(* CODESYS project testPrj.project
   Title: testPrj
   Version: 0.0.0.0

Project tree, tasks and I/O mapping:
  MyController : TM241CE40R, Schneider Electric, order no. TM241CE40R, version 4.0.2.20
    application Application
      libraries: Toolbox, 2.1.0.0 (Schneider Electric); Util, 3.5.1.0 (System)
      task MAST (freewheeling, priority 15, watchdog 100 ms x 1) calls main
      task Dempf (cyclic, interval t#50ms, priority 1) calls Analog
      function HiddenPOU [ST]
      global variables GVL
      Prog/
        program main [ST]
        program Analog [FBD]
    DI : Digital Inputs, Schneider Electric, version 4.0.2.20
        input  idwDI_IDW0 : DWORD  // IDW0
        input  Application.xDrumLH1 : BOOL  // IDW0.I0
        input  Application.xDrumLH2 : BOOL  // IDW0.I1
        input  Application.xDrumLl1 : BOOL  // IDW0.I2
        input  Application.xDrumLl2 : BOOL  // IDW0.I3
        input  Application.xFanRun : BOOL  // IDW0.I4
        input  Application.xExhRun : BOOL  // IDW0.I5
        input  Application.xPumpRun : BOOL  // IDW0.I6
        input  Application.xSafeOn : BOOL  // IDW0.I7
        input  Application.xDrumPh : BOOL  // IDW0.I8
        input  Application.xGasPl : BOOL  // IDW0.I9
        input  Application.xGasPh : BOOL  // IDW0.I10
        input  Application.xAirPl : BOOL  // IDW0.I11
        input  Application.xVacPl : BOOL  // IDW0.I12
        input  Application.xBump : BOOL  // IDW0.I13
        input  Application.xFire1 : BOOL  // IDW0.I14
        input  Application.xTight : BOOL  // IDW0.I15
        input  Application.xStartBn : BOOL  // IDW0.I16
        input  Application.xStopBn : BOOL  // IDW0.I17
        input  Application.xAlarmBn : BOOL  // IDW0.I18
        input  Application.xGasAuto : BOOL  // IDW0.I19
        input  Application.xTempAuto : BOOL  // IDW0.I20
        input  Application.xPumpAuto : BOOL  // IDW0.I21
        input  Application.xExhAuto : BOOL  // IDW0.I22
        input  Application.xFanAuto : BOOL  // IDW0.I23
        input  ibDI_IB1 : BYTE  // IB1
    DQ : Digital Outputs, Schneider Electric, version 4.0.2.20
        output Application.yCutofVal : BOOL  // QW0.Q0
        output Application.yBurnerVal : BOOL  // QW0.Q1
        output Application.ySafeVal : BOOL  // QW0.Q2
        output Application.yLitherVal : BOOL  // QW0.Q3
        output Application.yIgniter : BOOL  // QW0.Q4
        output Application.yStartFan : BOOL  // QW0.Q5
        output Application.yStartPump : BOOL  // QW0.Q6
        output Application.yGasOpen : BOOL  // QW0.Q7
        output Application.yGasClose : BOOL  // QW0.Q8
        output Application.yTempOpen : BOOL  // QW0.Q9
        output Application.yTempClose : BOOL  // QW0.Q10
        output Application.ySupOpen : BOOL  // QW0.Q11
        output Application.ySupClose : BOOL  // QW0.Q12
        output Application.yPlcStop : BOOL  // QW0.Q13
        output Application.ySerena : BOOL  // QW0.Q14
        output Application.yLamp : BOOL  // QW0.Q15
        output qbDQ_QB1 : BYTE  // QB1
        unmapped channels: QW0
    Counters : Counters, Schneider Electric, version 4.0.2.20
    Pulse_Generators : Pulse Generators, Schneider Electric, version 4.0.2.20
    Cartridge_1 : Cartridge, Schneider Electric, version 4.0.2.20
    Cartridge_2 : Cartridge, Schneider Electric, version 4.0.2.20
    IO_Bus : IO bus - TM3, Schneider Electric, version 4.0.2.20
      Module_1 : TM3AQ4/G, Schneider Electric, order no. TM3AQ4/G, version 1.0.0.10
          settings: KPI Configuration.KPI Configuration[0] = 19; KPI Configuration.KPI Configuration[1] = 19; KPI Configuration.KPI Configuration[2] = 19; KPI Configuration.KPI Configuration[3] = 19; KPI Configuration.KPI Configuration[5] = 0; KPI Configuration.KPI Configuration[7] = 0; KPI Configuration.KPI Configuration[9] = 0; KPI Configuration.KPI Configuration[11] = 0; KPI Configuration.KPI Configuration[12] = 160; KPI Configuration.KPI Configuration[13] = 15; KPI Configuration.KPI Configuration[14] = 160; KPI Configuration.KPI Configuration[15] = 15; KPI Configuration.KPI Configuration[16] = 160; KPI Configuration.KPI Configuration[17] = 15; KPI Configuration.KPI Configuration[18] = 160; KPI Configuration.KPI Configuration[19] = 15
          output C0001 : INT  // QW0
          output C0002 : INT  // QW1
          output C0003 : INT  // QW2
          output C0004 : INT  // QW3
          input  ibModule_1_IBStatusQW0 : BYTE  // IBStatusQW0
          input  ibModule_1_IBStatusQW1 : BYTE  // IBStatusQW1
          input  ibModule_1_IBStatusQW2 : BYTE  // IBStatusQW2
          input  ibModule_1_IBStatusQW3 : BYTE  // IBStatusQW3
      Module_2 : TM3AI8/G, Schneider Electric, order no. TM3AI8/G, version 1.0.0.12
          settings: KPI Configuration.KPI Configuration[0] = 35; KPI Configuration.KPI Configuration[1] = 35; KPI Configuration.KPI Configuration[2] = 35; KPI Configuration.KPI Configuration[3] = 35; KPI Configuration.KPI Configuration[4] = 35; KPI Configuration.KPI Configuration[5] = 35; KPI Configuration.KPI Configuration[6] = 35; KPI Configuration.KPI Configuration[7] = 35; KPI Configuration.KPI Configuration[9] = 0; KPI Configuration.KPI Configuration[11] = 0; KPI Configuration.KPI Configuration[13] = 0; KPI Configuration.KPI Configuration[15] = 0; KPI Configuration.KPI Configuration[17] = 0; KPI Configuration.KPI Configuration[19] = 0; KPI Configuration.KPI Configuration[21] = 0; KPI Configuration.KPI Configuration[23] = 0; KPI Configuration.KPI Configuration[24] = 160; KPI Configuration.KPI Configuration[25] = 15; KPI Configuration.KPI Configuration[26] = 160; KPI Configuration.KPI Configuration[27] = 15; KPI Configuration.KPI Configuration[28] = 160; KPI Configuration.KPI Configuration[29] = 15; KPI Configuration.KPI Configuration[30] = 160; KPI Configuration.KPI Configuration[31] = 15; KPI Configuration.KPI Configuration[32] = 160; KPI Configuration.KPI Configuration[33] = 15; KPI Configuration.KPI Configuration[34] = 160; KPI Configuration.KPI Configuration[35] = 15; KPI Configuration.KPI Configuration[36] = 160; KPI Configuration.KPI Configuration[37] = 15; KPI Configuration.KPI Configuration[38] = 160; KPI Configuration.KPI Configuration[39] = 15
          input  A0000 : INT  // IW0
          input  A0001 : INT  // IW1
          input  A0002 : INT  // IW2
          input  A0003 : INT  // IW3
          input  A0004 : INT  // IW4
          input  A0005 : INT  // IW5
          input  A0006 : INT  // IW6
          input  A0007 : INT  // IW7
          input  ibModule_2_IBStatusIW0 : BYTE  // IBStatusIW0
          input  ibModule_2_IBStatusIW1 : BYTE  // IBStatusIW1
          input  ibModule_2_IBStatusIW2 : BYTE  // IBStatusIW2
          input  ibModule_2_IBStatusIW3 : BYTE  // IBStatusIW3
          input  ibModule_2_IBStatusIW4 : BYTE  // IBStatusIW4
          input  ibModule_2_IBStatusIW5 : BYTE  // IBStatusIW5
          input  ibModule_2_IBStatusIW6 : BYTE  // IBStatusIW6
          input  ibModule_2_IBStatusIW7 : BYTE  // IBStatusIW7
      Module_3 : TM3AI8/G, Schneider Electric, order no. TM3AI8/G, version 1.0.0.12
          settings: KPI Configuration.KPI Configuration[0] = 35; KPI Configuration.KPI Configuration[1] = 35; KPI Configuration.KPI Configuration[2] = 35; KPI Configuration.KPI Configuration[3] = 35; KPI Configuration.KPI Configuration[4] = 35; KPI Configuration.KPI Configuration[5] = 35; KPI Configuration.KPI Configuration[6] = 35; KPI Configuration.KPI Configuration[7] = 35; KPI Configuration.KPI Configuration[9] = 0; KPI Configuration.KPI Configuration[11] = 0; KPI Configuration.KPI Configuration[13] = 0; KPI Configuration.KPI Configuration[15] = 0; KPI Configuration.KPI Configuration[17] = 0; KPI Configuration.KPI Configuration[19] = 0; KPI Configuration.KPI Configuration[21] = 0; KPI Configuration.KPI Configuration[23] = 0; KPI Configuration.KPI Configuration[24] = 160; KPI Configuration.KPI Configuration[25] = 15; KPI Configuration.KPI Configuration[26] = 160; KPI Configuration.KPI Configuration[27] = 15; KPI Configuration.KPI Configuration[28] = 160; KPI Configuration.KPI Configuration[29] = 15; KPI Configuration.KPI Configuration[30] = 160; KPI Configuration.KPI Configuration[31] = 15; KPI Configuration.KPI Configuration[32] = 160; KPI Configuration.KPI Configuration[33] = 15; KPI Configuration.KPI Configuration[34] = 160; KPI Configuration.KPI Configuration[35] = 15; KPI Configuration.KPI Configuration[36] = 232; KPI Configuration.KPI Configuration[37] = 3; KPI Configuration.KPI Configuration[38] = 160; KPI Configuration.KPI Configuration[39] = 15
          input  A0010 : INT  // IW0
          input  A0011 : INT  // IW1
          input  A0012 : INT  // IW2
          input  A0013 : INT  // IW3
          input  A0014 : INT  // IW4
          input  A0015 : INT  // IW5
          input  A0016 : INT  // IW6
          input  A0017 : INT  // IW7
          input  ibModule_3_IBStatusIW0 : BYTE  // IBStatusIW0
          input  ibModule_3_IBStatusIW1 : BYTE  // IBStatusIW1
          input  ibModule_3_IBStatusIW2 : BYTE  // IBStatusIW2
          input  ibModule_3_IBStatusIW3 : BYTE  // IBStatusIW3
          input  ibModule_3_IBStatusIW4 : BYTE  // IBStatusIW4
          input  ibModule_3_IBStatusIW5 : BYTE  // IBStatusIW5
          input  ibModule_3_IBStatusIW6 : BYTE  // IBStatusIW6
          input  ibModule_3_IBStatusIW7 : BYTE  // IBStatusIW7
      Module_4 : TM3AI8/G, Schneider Electric, order no. TM3AI8/G, version 1.0.0.12
          settings: KPI Configuration.KPI Configuration[0] = 35; KPI Configuration.KPI Configuration[1] = 35; KPI Configuration.KPI Configuration[2] = 35; KPI Configuration.KPI Configuration[3] = 35; KPI Configuration.KPI Configuration[4] = 35; KPI Configuration.KPI Configuration[5] = 35; KPI Configuration.KPI Configuration[6] = 35; KPI Configuration.KPI Configuration[7] = 35; KPI Configuration.KPI Configuration[9] = 0; KPI Configuration.KPI Configuration[11] = 0; KPI Configuration.KPI Configuration[13] = 0; KPI Configuration.KPI Configuration[15] = 0; KPI Configuration.KPI Configuration[17] = 0; KPI Configuration.KPI Configuration[19] = 0; KPI Configuration.KPI Configuration[21] = 0; KPI Configuration.KPI Configuration[23] = 0; KPI Configuration.KPI Configuration[24] = 160; KPI Configuration.KPI Configuration[25] = 15; KPI Configuration.KPI Configuration[26] = 160; KPI Configuration.KPI Configuration[27] = 15; KPI Configuration.KPI Configuration[28] = 160; KPI Configuration.KPI Configuration[29] = 15; KPI Configuration.KPI Configuration[30] = 160; KPI Configuration.KPI Configuration[31] = 15; KPI Configuration.KPI Configuration[32] = 160; KPI Configuration.KPI Configuration[33] = 15; KPI Configuration.KPI Configuration[34] = 160; KPI Configuration.KPI Configuration[35] = 15; KPI Configuration.KPI Configuration[36] = 160; KPI Configuration.KPI Configuration[37] = 15; KPI Configuration.KPI Configuration[38] = 160; KPI Configuration.KPI Configuration[39] = 15
          input  A0020 : INT  // IW0
          input  A0021 : INT  // IW1
          input  A0022 : INT  // IW2
          input  A0023 : INT  // IW3
          input  A0024 : INT  // IW4
          input  A0025 : INT  // IW5
          input  A0026 : INT  // IW6
          input  A0027 : INT  // IW7
          input  ibModule_4_IBStatusIW0 : BYTE  // IBStatusIW0
          input  ibModule_4_IBStatusIW1 : BYTE  // IBStatusIW1
          input  ibModule_4_IBStatusIW2 : BYTE  // IBStatusIW2
          input  ibModule_4_IBStatusIW3 : BYTE  // IBStatusIW3
          input  ibModule_4_IBStatusIW4 : BYTE  // IBStatusIW4
          input  ibModule_4_IBStatusIW5 : BYTE  // IBStatusIW5
          input  ibModule_4_IBStatusIW6 : BYTE  // IBStatusIW6
          input  ibModule_4_IBStatusIW7 : BYTE  // IBStatusIW7
    COM_Bus : COM bus, Schneider Electric, version 4.0.2.20
    Ethernet_1 : Ethernet Network, Schneider Electric, version 4.0.2.20
        settings: IPAddress = [192, 168, 15, 152]; SubnetMask = [255, 255, 255, 0]; GatewayAddress = [192, 168, 15, 1]; WebServer = FALSE; FTP Server = FALSE; SoMachine Protocol = TRUE; Modbus Server = TRUE; NetManage Protocol = FALSE; SNMP protocol = FALSE; Enable Routing = FALSE; WebVisu protocol = FALSE
      ModbusTCP_Slave_Device : ModbusTCP Slave Device, Schneider Electric, version 3.5.2.3
          unmapped channels: Inputs, Outputs
    Serial_Line_1 : Serial line, Schneider Electric, version 4.0.2.20
    Serial_Line_2 : Serial line, Schneider Electric, version 4.0.2.20
      Modbus_IOScanner : Modbus IOScanner, Schneider Electric, version 3.5.3.6
        Generic_Modbus_Slave : Generic Modbus Slave, Schneider Electric, version 3.5.3.6
            settings: Channel 1.Function Code = 3; Channel 1.Read Offset = 16#1001; Channel 1.Read Length = 6; Channel 1.Write Offset = 0; Channel 1.Write Length = 0; Channel 1.Cycle Time = 100; Channel 2.Function Code = 3; Channel 2.Read Offset = 16#8000; Channel 2.Read Length = 1; Channel 2.Write Offset = 0; Channel 2.Write Length = 0; Channel 2.Cycle Time = 100; Channel 3.Function Code = 3; Channel 3.Read Offset = 16#3000; Channel 3.Read Length = 1; Channel 3.Write Offset = 0; Channel 3.Write Length = 0; Channel 3.Cycle Time = 100
            input  M1 : WORD  // Channel 1.Channel 1[0]
            input  M2 : WORD  // Channel 1.Channel 1[1]
            input  M3 : WORD  // Channel 1.Channel 1[2]
            input  M4 : WORD  // Channel 1.Channel 1[3]
            input  M5 : WORD  // Channel 1.Channel 1[4]
            input  M6 : WORD  // Channel 1.Channel 1[5]
            input  M7 : WORD  // Channel 2.Channel 2[0]
            input  M8 : WORD  // Channel 3.Channel 3[0]
            unmapped channels: Channel 1, Channel 2, Channel 3
*)

// MyController/Application/GVL
VAR_GLOBAL

Run AT %M9: BOOL;

xDrumLH1 AT %M10: BOOL;
xDrumLH2 AT %M11: BOOL;
xDrumLl1 AT %M12: BOOL;
xDrumLl2 AT %M13: BOOL;
xFanRun AT %M14: BOOL;
xExhRun AT %M15: BOOL;
xPumpRun AT %M16: BOOL;
xSafeOn AT %M17: BOOL;
xDrumPh AT %M18: BOOL;
xGasPl AT %M19: BOOL;
xGasPh AT %M20: BOOL;
xAirPl AT %M21: BOOL;
xVacPl AT %M22: BOOL;
xBump AT %M23: BOOL;
xFire1 AT %M24: BOOL;
xTight AT %M25: BOOL;
xStartBn AT %M26: BOOL;
xStopBn AT %M27: BOOL;
xAlarmBn AT %M28: BOOL;
xGasAuto AT %M29: BOOL;
xTempAuto AT %M30: BOOL;
xPumpAuto AT %M31: BOOL;
xExhAuto AT %M32: BOOL;
xFanAuto AT %M33: BOOL;

yCutofVal AT %M34: BOOL;
yBurnerVal AT %M35: BOOL;
ySafeVal AT %M36: BOOL;
yLitherVal AT %M37: BOOL;
yIgniter AT %M38: BOOL;
yStartFan AT %M39: BOOL;
yStartPump AT %M40: BOOL;
yGasOpen AT %M41: BOOL;
yGasClose AT %M42: BOOL;
yTempOpen AT %M43: BOOL;
yTempClose AT %M44: BOOL;
ySupOpen AT %M45: BOOL;
ySupClose AT %M46: BOOL;
yPlcStop AT %M47: BOOL;
ySerena AT %M48: BOOL;
yLamp AT %M49: BOOL;

Fg AT %MD9: REAL;
Fp AT %MD11: REAL;
Fv AT %MD13: REAL;
Fa AT %MD15: REAL;
Lv AT %MD17: REAL;
Tpar AT %MD19: REAL;
Tv3a AT %MD21: REAL;
Tv4a AT %MD23: REAL;
Tk AT %MD25: REAL;
Ta5a AT %MD27: REAL;
Ta6a AT %MD29: REAL;
Tp17a AT %MD31: REAL;
Tp18a AT %MD33: REAL;
Pg15a AT %MD35: REAL;
Pp AT %MD37: REAL;
Pp7a AT %MD39: REAL;
Pa AT %MD41: REAL;
Pv AT %MD43: REAL;
Pv12a AT %MD45: REAL;
Gg AT %MD47: REAL;
Gph AT %MD49: REAL;
Gpc AT %MD51: REAL;
Qa AT %MD53: REAL;
Vx AT %MD55: REAL;
Cv AT %MD57: REAL;
Cp AT %MD59: REAL;
Ca AT %MD61: REAL;
Cx AT %MD63: REAL;

fA0000 AT %MW65: UINT;
fA0001 AT %MW66: UINT;
fA0002 AT %MW67: UINT;
fA0003 AT %MW68: UINT;
fA0004 AT %MW69: UINT;
fA0005 AT %MW70: UINT;
fA0006 AT %MW71: UINT;
fA0007 AT %MW72: UINT;
fA0010 AT %MW73: UINT;
fA0011 AT %MW74: UINT;
fA0012 AT %MW75: UINT;
fA0013 AT %MW76: UINT;
fA0014 AT %MW77: UINT;
fA0015 AT %MW78: UINT;
fA0016 AT %MW79: UINT;
fA0017 AT %MW80: UINT;
fA0020 AT %MW81: UINT;
fA0021 AT %MW82: UINT;
fA0022 AT %MW83: UINT;
fA0023 AT %MW84: UINT;
fA0024 AT %MW85: UINT;
fA0025 AT %MW86: UINT;
fA0026 AT %MW87: UINT;
fA0027 AT %MW88: UINT;


END_VAR

// MyController/Application/Prog/main
PROGRAM main
VAR
END_VAR

END_PROGRAM

// MyController/Application/Prog/Analog
PROGRAM Analog
VAR
avg0000: SE_TBX.Filter_MovingAverage;
avg0001: SE_TBX.Filter_MovingAverage;
avg0002: SE_TBX.Filter_MovingAverage;
avg0003: SE_TBX.Filter_MovingAverage;
avg0004: SE_TBX.Filter_MovingAverage;
avg0005: SE_TBX.Filter_MovingAverage;
avg0006: SE_TBX.Filter_MovingAverage;
avg0007: SE_TBX.Filter_MovingAverage;
avg0010: SE_TBX.Filter_MovingAverage;
avg0011: SE_TBX.Filter_MovingAverage;
avg0012: SE_TBX.Filter_MovingAverage;
avg0013: SE_TBX.Filter_MovingAverage;
avg0014: SE_TBX.Filter_MovingAverage;
avg0015: SE_TBX.Filter_MovingAverage;
avg0016: SE_TBX.Filter_MovingAverage;
avg0017: SE_TBX.Filter_MovingAverage;
avg0020: SE_TBX.Filter_MovingAverage;
avg0021: SE_TBX.Filter_MovingAverage;
avg0022: SE_TBX.Filter_MovingAverage;
avg0023: SE_TBX.Filter_MovingAverage;
avg0024: SE_TBX.Filter_MovingAverage;
avg0025: SE_TBX.Filter_MovingAverage;
avg0026: SE_TBX.Filter_MovingAverage;
avg0027: SE_TBX.Filter_MovingAverage;

END_VAR
VAR
END_VAR
VAR // added by the converter: edge detectors and wires of the graphical bodies
    _rt1, _rt2, _rt3, _rt4, _rt5, _rt6, _rt7, _rt8, _rt9, _rt10, _rt11, _rt12, _rt13, _rt14, _rt15, _rt16, _rt17, _rt18, _rt19, _rt20, _rt21, _rt22, _rt23, _rt24 : R_TRIG;
END_VAR

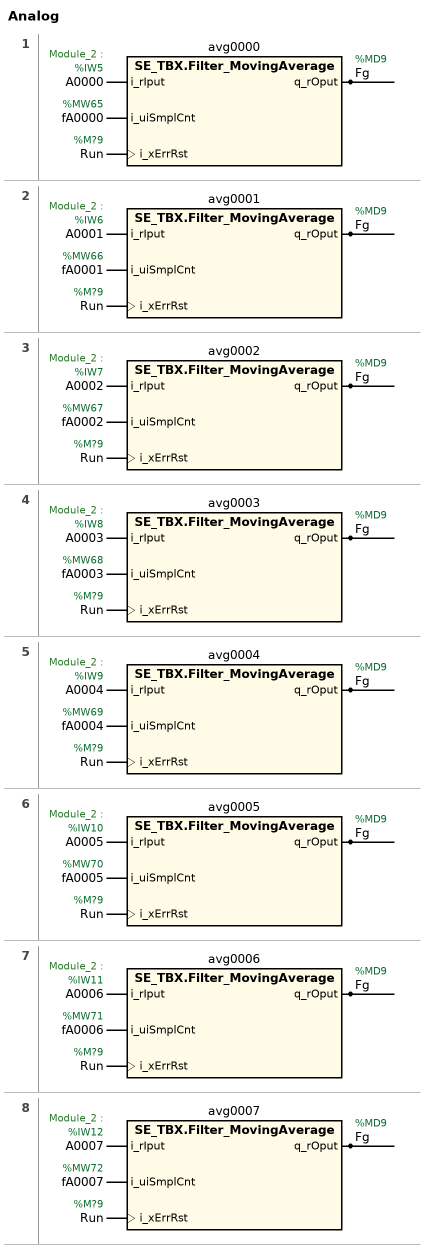
// NETWORK 1
//   A0000: Module_2 : | AT %IW5
//   fA0000: AT %MW65
//   Run: AT %M?9
//   Fg: AT %MD9
_rt1(CLK := Run);
avg0000(i_rIput := A0000, i_uiSmplCnt := fA0000, i_xErrRst := _rt1.Q, q_rOput => Fg); // SE_TBX.Filter_MovingAverage

// NETWORK 2
//   A0001: Module_2 : | AT %IW6
//   fA0001: AT %MW66
//   Run: AT %M?9
//   Fg: AT %MD9
_rt2(CLK := Run);
avg0001(i_rIput := A0001, i_uiSmplCnt := fA0001, i_xErrRst := _rt2.Q, q_rOput => Fg); // SE_TBX.Filter_MovingAverage

// NETWORK 3
//   A0002: Module_2 : | AT %IW7
//   fA0002: AT %MW67
//   Run: AT %M?9
//   Fg: AT %MD9
_rt3(CLK := Run);
avg0002(i_rIput := A0002, i_uiSmplCnt := fA0002, i_xErrRst := _rt3.Q, q_rOput => Fg); // SE_TBX.Filter_MovingAverage

// NETWORK 4
//   A0003: Module_2 : | AT %IW8
//   fA0003: AT %MW68
//   Run: AT %M?9
//   Fg: AT %MD9
_rt4(CLK := Run);
avg0003(i_rIput := A0003, i_uiSmplCnt := fA0003, i_xErrRst := _rt4.Q, q_rOput => Fg); // SE_TBX.Filter_MovingAverage

// NETWORK 5
//   A0004: Module_2 : | AT %IW9
//   fA0004: AT %MW69
//   Run: AT %M?9
//   Fg: AT %MD9
_rt5(CLK := Run);
avg0004(i_rIput := A0004, i_uiSmplCnt := fA0004, i_xErrRst := _rt5.Q, q_rOput => Fg); // SE_TBX.Filter_MovingAverage

// NETWORK 6
//   A0005: Module_2 : | AT %IW10
//   fA0005: AT %MW70
//   Run: AT %M?9
//   Fg: AT %MD9
_rt6(CLK := Run);
avg0005(i_rIput := A0005, i_uiSmplCnt := fA0005, i_xErrRst := _rt6.Q, q_rOput => Fg); // SE_TBX.Filter_MovingAverage

// NETWORK 7
//   A0006: Module_2 : | AT %IW11
//   fA0006: AT %MW71
//   Run: AT %M?9
//   Fg: AT %MD9
_rt7(CLK := Run);
avg0006(i_rIput := A0006, i_uiSmplCnt := fA0006, i_xErrRst := _rt7.Q, q_rOput => Fg); // SE_TBX.Filter_MovingAverage

// NETWORK 8
//   A0007: Module_2 : | AT %IW12
//   fA0007: AT %MW72
//   Run: AT %M?9
//   Fg: AT %MD9
_rt8(CLK := Run);
avg0007(i_rIput := A0007, i_uiSmplCnt := fA0007, i_xErrRst := _rt8.Q, q_rOput => Fg); // SE_TBX.Filter_MovingAverage

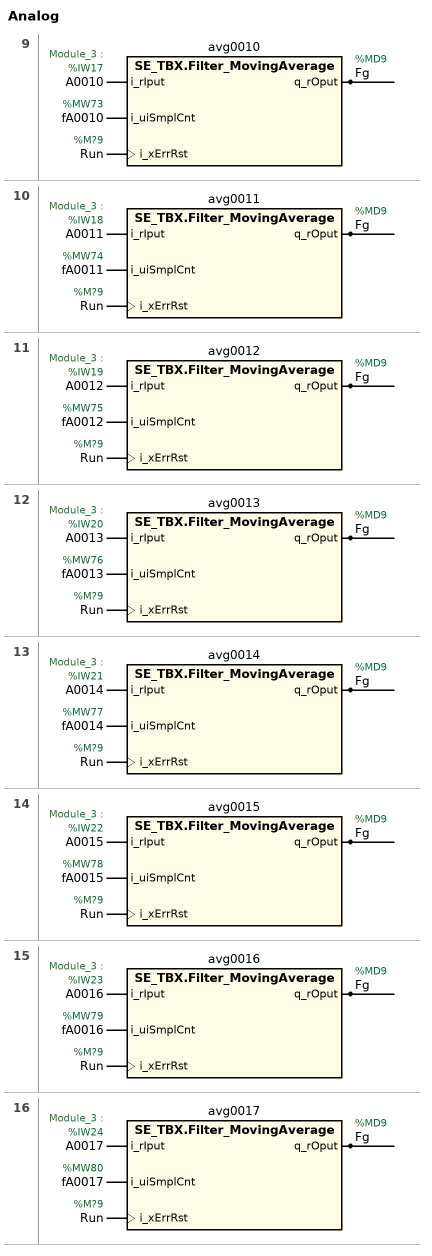
// NETWORK 9
//   A0010: Module_3 : | AT %IW17
//   fA0010: AT %MW73
//   Run: AT %M?9
//   Fg: AT %MD9
_rt9(CLK := Run);
avg0010(i_rIput := A0010, i_uiSmplCnt := fA0010, i_xErrRst := _rt9.Q, q_rOput => Fg); // SE_TBX.Filter_MovingAverage

// NETWORK 10
//   A0011: Module_3 : | AT %IW18
//   fA0011: AT %MW74
//   Run: AT %M?9
//   Fg: AT %MD9
_rt10(CLK := Run);
avg0011(i_rIput := A0011, i_uiSmplCnt := fA0011, i_xErrRst := _rt10.Q, q_rOput => Fg); // SE_TBX.Filter_MovingAverage

// NETWORK 11
//   A0012: Module_3 : | AT %IW19
//   fA0012: AT %MW75
//   Run: AT %M?9
//   Fg: AT %MD9
_rt11(CLK := Run);
avg0012(i_rIput := A0012, i_uiSmplCnt := fA0012, i_xErrRst := _rt11.Q, q_rOput => Fg); // SE_TBX.Filter_MovingAverage

// NETWORK 12
//   A0013: Module_3 : | AT %IW20
//   fA0013: AT %MW76
//   Run: AT %M?9
//   Fg: AT %MD9
_rt12(CLK := Run);
avg0013(i_rIput := A0013, i_uiSmplCnt := fA0013, i_xErrRst := _rt12.Q, q_rOput => Fg); // SE_TBX.Filter_MovingAverage

// NETWORK 13
//   A0014: Module_3 : | AT %IW21
//   fA0014: AT %MW77
//   Run: AT %M?9
//   Fg: AT %MD9
_rt13(CLK := Run);
avg0014(i_rIput := A0014, i_uiSmplCnt := fA0014, i_xErrRst := _rt13.Q, q_rOput => Fg); // SE_TBX.Filter_MovingAverage

// NETWORK 14
//   A0015: Module_3 : | AT %IW22
//   fA0015: AT %MW78
//   Run: AT %M?9
//   Fg: AT %MD9
_rt14(CLK := Run);
avg0015(i_rIput := A0015, i_uiSmplCnt := fA0015, i_xErrRst := _rt14.Q, q_rOput => Fg); // SE_TBX.Filter_MovingAverage

// NETWORK 15
//   A0016: Module_3 : | AT %IW23
//   fA0016: AT %MW79
//   Run: AT %M?9
//   Fg: AT %MD9
_rt15(CLK := Run);
avg0016(i_rIput := A0016, i_uiSmplCnt := fA0016, i_xErrRst := _rt15.Q, q_rOput => Fg); // SE_TBX.Filter_MovingAverage

// NETWORK 16
//   A0017: Module_3 : | AT %IW24
//   fA0017: AT %MW80
//   Run: AT %M?9
//   Fg: AT %MD9
_rt16(CLK := Run);
avg0017(i_rIput := A0017, i_uiSmplCnt := fA0017, i_xErrRst := _rt16.Q, q_rOput => Fg); // SE_TBX.Filter_MovingAverage

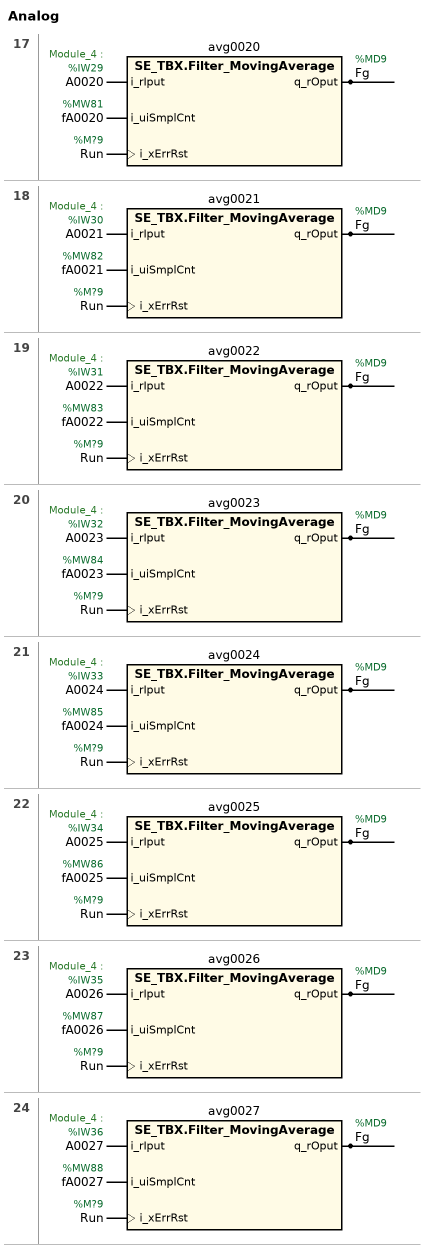
// NETWORK 17
//   A0020: Module_4 : | AT %IW29
//   fA0020: AT %MW81
//   Run: AT %M?9
//   Fg: AT %MD9
_rt17(CLK := Run);
avg0020(i_rIput := A0020, i_uiSmplCnt := fA0020, i_xErrRst := _rt17.Q, q_rOput => Fg); // SE_TBX.Filter_MovingAverage

// NETWORK 18
//   A0021: Module_4 : | AT %IW30
//   fA0021: AT %MW82
//   Run: AT %M?9
//   Fg: AT %MD9
_rt18(CLK := Run);
avg0021(i_rIput := A0021, i_uiSmplCnt := fA0021, i_xErrRst := _rt18.Q, q_rOput => Fg); // SE_TBX.Filter_MovingAverage

// NETWORK 19
//   A0022: Module_4 : | AT %IW31
//   fA0022: AT %MW83
//   Run: AT %M?9
//   Fg: AT %MD9
_rt19(CLK := Run);
avg0022(i_rIput := A0022, i_uiSmplCnt := fA0022, i_xErrRst := _rt19.Q, q_rOput => Fg); // SE_TBX.Filter_MovingAverage

// NETWORK 20
//   A0023: Module_4 : | AT %IW32
//   fA0023: AT %MW84
//   Run: AT %M?9
//   Fg: AT %MD9
_rt20(CLK := Run);
avg0023(i_rIput := A0023, i_uiSmplCnt := fA0023, i_xErrRst := _rt20.Q, q_rOput => Fg); // SE_TBX.Filter_MovingAverage

// NETWORK 21
//   A0024: Module_4 : | AT %IW33
//   fA0024: AT %MW85
//   Run: AT %M?9
//   Fg: AT %MD9
_rt21(CLK := Run);
avg0024(i_rIput := A0024, i_uiSmplCnt := fA0024, i_xErrRst := _rt21.Q, q_rOput => Fg); // SE_TBX.Filter_MovingAverage

// NETWORK 22
//   A0025: Module_4 : | AT %IW34
//   fA0025: AT %MW86
//   Run: AT %M?9
//   Fg: AT %MD9
_rt22(CLK := Run);
avg0025(i_rIput := A0025, i_uiSmplCnt := fA0025, i_xErrRst := _rt22.Q, q_rOput => Fg); // SE_TBX.Filter_MovingAverage

// NETWORK 23
//   A0026: Module_4 : | AT %IW35
//   fA0026: AT %MW87
//   Run: AT %M?9
//   Fg: AT %MD9
_rt23(CLK := Run);
avg0026(i_rIput := A0026, i_uiSmplCnt := fA0026, i_xErrRst := _rt23.Q, q_rOput => Fg); // SE_TBX.Filter_MovingAverage

// NETWORK 24
//   A0027: Module_4 : | AT %IW36
//   fA0027: AT %MW88
//   Run: AT %M?9
//   Fg: AT %MD9
_rt24(CLK := Run);
avg0027(i_rIput := A0027, i_uiSmplCnt := fA0027, i_xErrRst := _rt24.Q, q_rOput => Fg); // SE_TBX.Filter_MovingAverage

END_PROGRAM

// MyController/Application/HiddenPOU
FUNCTION HiddenPOU : BOOL

VAR_INPUT
	pHiddenFunc: POINTER TO WORD;
END_VAR
VAR
	pRead: POINTER TO BYTE;
	pWrite: POINTER TO BYTE;
END_VAR

pRead := pHiddenFunc + 400;
pWrite := pHiddenFunc + 4400;
HiddenPOU := TRUE;

END_FUNCTION
